// TIA Portal V20 export
DATA_BLOCK "HardwareIO"   // DB8
{ S7_Optimized_Access := 'TRUE' }
// stored: MemoryReserve 100
   VAR
      DigitalInputs : Struct
         DI001_Input : Bool;
         VSD001_ForewardFB : Bool;
         VSD001_ReverseFB : Bool;
         VSD001_TripFB : Bool;
         MOT001_ForewardFB : Bool;
         MOT001_ReverseFB : Bool;
         MOT001_TripFB : Bool;
         VLV001_OpenFB : Bool;
         VLV001_ClosedFB : Bool;
         VLV001_Fault : Bool;
         CONTVLV001_OpenFB : Bool;
         CONTVLV001_ClosedFB : Bool;
         CONTVLV001_Fault : Bool;
      END_STRUCT;
      DigitalOutputs : Struct
         DO001_Output : Bool;
         VSD001_ForwardCmd : Bool;
         VSD001_ReverseCmd : Bool;
         MOT001_ForwardCmd : Bool;
         MOT001_ReverseCmd : Bool;
         VLV001_OpenCmd : Bool;
         VLV001_CloseCmd : Bool;
         CONTVLV001_OpenCmd : Bool;
         CONTVLV001_CloseCmd : Bool;
      END_STRUCT;
      AnalogueInputs : Struct
         AI001_Value : Real;
         VSD001_SpeedFB : Real;
         CONTVLV001_PositionFB : Real;
      END_STRUCT;
      AnalogueOutputs : Struct
         AO001_Value : Real;
         VSD001_SpeedCmd : Real;
         CONTVLV001_PositionCmd : Real;
      END_STRUCT;
   END_VAR
BEGIN
END_DATA_BLOCK
